{attribute 'qualified_only'}
{attribute 'strict'}
TYPE INTERNAL eMessageCondition :
(
    Unconditional := 0,
    Active := 10,
    Inactive := 20
);
END_TYPE

(* stored: Version 1.1.0.1
   DUT eMessageCondition: Id {39702f60-a703-05b9-36f5-1f05c6331443} *)
